{attribute addProperty BoxType "EK1122-0000-0018"}
{attribute addProperty Id "Beckhoff_EPP1xxxsub_EK1100EK1100_179A0949162A_0001_EPP1004_0061_0016EPP1004_C1DCB3BD506.25A_0002_EPP1008_0001_0016EPP1008_772BB4148210.25A_0003_EPP1008_0001_0017EPP1008_772BB4148210.25A_0004_EPP1008_0002_0016EPP1008_772BB4148210.25A_0005_EPP1008_0002_0017EPP1008_772BB4148210.25A_0006_EPP1008_0022_0016EPP1008_772BB4148210.25A_0007_EPP1018_0001_0016EPP1018_772BB4148210.25A_0008_EPP1018_0001_0017EPP1018_772BB4148210.25A_0009_EPP1018_0002_0016EPP1018_772BB4148210.25A_0010_EPP1018_0002_0017EPP1018_772BB4148210.25A_0011_EPP1111_0000_0016EPP1111_0792AF759812.25A_0012_EPP1111_0000_0017EPP1111_0792AF759812.25A_0013_EPP1111_0000_0018EPP1111_0792AF759812.25A_0014_EPP1258_0001_0016EPP1258_BB8E9A1042052.5A_0015_EPP1258_0001_0017EPP1258_BB8E9A1042052.5A_0016_EPP1258_0002_0016EPP1258_BB8E9A1042052.5A_0017_EPP1258_0002_0017EPP1258_BB8E9A1042052.5A_0018_EPP1321_0060_0016A_0018_EPP1321_0060_0016_CF61AE2B2662332.75"}
{attribute addProperty CRC "3483081605"}
{attribute addProperty SizeInBites "5440"}
{attribute addProperty SizeInBytes "680"}
TYPE Beckhoff_EPP1xxxEK1122_CF9B9B85 EXTENDS EK1122_179A0949 :
STRUCT
	{attribute addProperty Name "Beckhoff_EPP1xxxsub_EK1100"}
	Beckhoff_EPP1xxxsub_EK1100 : EK1100_179A0949;
	{attribute addProperty Name "A_0001_EPP1004_0061_0016"}
	A_0001_EPP1004_0061_0016 : EPP1004_C1DCB3BD;
	{attribute addProperty Name "A_0002_EPP1008_0001_0016"}
	A_0002_EPP1008_0001_0016 : EPP1008_772BB414;
	{attribute addProperty Name "A_0003_EPP1008_0001_0017"}
	A_0003_EPP1008_0001_0017 : EPP1008_772BB414;
	{attribute addProperty Name "A_0004_EPP1008_0002_0016"}
	A_0004_EPP1008_0002_0016 : EPP1008_772BB414;
	{attribute addProperty Name "A_0005_EPP1008_0002_0017"}
	A_0005_EPP1008_0002_0017 : EPP1008_772BB414;
	{attribute addProperty Name "A_0006_EPP1008_0022_0016"}
	A_0006_EPP1008_0022_0016 : EPP1008_772BB414;
	{attribute addProperty Name "A_0007_EPP1018_0001_0016"}
	A_0007_EPP1018_0001_0016 : EPP1018_772BB414;
	{attribute addProperty Name "A_0008_EPP1018_0001_0017"}
	A_0008_EPP1018_0001_0017 : EPP1018_772BB414;
	{attribute addProperty Name "A_0009_EPP1018_0002_0016"}
	A_0009_EPP1018_0002_0016 : EPP1018_772BB414;
	{attribute addProperty Name "A_0010_EPP1018_0002_0017"}
	A_0010_EPP1018_0002_0017 : EPP1018_772BB414;
	{attribute addProperty Name "A_0011_EPP1111_0000_0016"}
	A_0011_EPP1111_0000_0016 : EPP1111_0792AF75;
	{attribute addProperty Name "A_0012_EPP1111_0000_0017"}
	A_0012_EPP1111_0000_0017 : EPP1111_0792AF75;
	{attribute addProperty Name "A_0013_EPP1111_0000_0018"}
	A_0013_EPP1111_0000_0018 : EPP1111_0792AF75;
	{attribute addProperty Name "A_0014_EPP1258_0001_0016"}
	A_0014_EPP1258_0001_0016 : EPP1258_BB8E9A10;
	{attribute addProperty Name "A_0015_EPP1258_0001_0017"}
	A_0015_EPP1258_0001_0017 : EPP1258_BB8E9A10;
	{attribute addProperty Name "A_0016_EPP1258_0002_0016"}
	A_0016_EPP1258_0002_0016 : EPP1258_BB8E9A10;
	{attribute addProperty Name "A_0017_EPP1258_0002_0017"}
	A_0017_EPP1258_0002_0017 : EPP1258_BB8E9A10;
	{attribute addProperty Name "A_0018_EPP1321_0060_0016"}
	A_0018_EPP1321_0060_0016 : A_0018_EPP1321_0060_0016_CF61AE2B;
END_STRUCT
END_TYPE

(* stored: Version 1.2.0.0, ProductVersion 3.1.4024.9
   DUT Beckhoff_EPP1xxxEK1122_CF9B9B85: Id {97022419-01d9-4b59-be8e-4df64e5bcf70} *)
